Fanuc KAREL source: kt00007.KL

-- PROVISIONAL review KL for V1013-1; original PC SHA256 7edf0f945f1a272328144f80028967fdadfb95a9e5e862af6eb83b4927aa437c
-- Incomplete behavior may be omitted. Consult companion uncertainty JSON. Do not deploy.
PROGRAM KT00007
%NOLOCKGROUP
VAR
  I1 : INTEGER
  OUT : INTEGER
-- UNRESOLVED_DECL H2 type=002017
BEGIN
  -- UNRESOLVED_PC offsets 5-16; opcodes 2E,23
  -- UNRESOLVED_PC offsets 21-35; opcodes 2E,22,9D,33,B4
  -- UNRESOLVED_PC offsets 40-62; opcodes 21,22,9D,33,B3,52,23
  -- UNRESOLVED_PC offsets 67-71; opcodes 7F
END KT00007
